// TIA Portal project "Travail_2_station_pince" (V19)

(* hardware
DEVICE "S7-300/ET200M station_1"  S7-300 station
   slot 0: "Rail_0"  Rail  6ES7 390-1***0-0AA0
   slot 2: "PLC_1"  CPU 314C-2 PN/DP  6ES7 314-6EH04-0AB0  V3.3
      slot 2: "PROFINET interface_1"  PN-IO
         slot 1: "Port_1"  Port
         slot 2: "Port_2"  Port
      slot 5: "DI 24/DO 16_1"  DI24/DO16
      slot 6: "AI 5/AO 2_1"  AI5/AO2
      slot 7: "Count_1"  Counter
      slot 8: "Positioning_1"  Positioning
*)

// ===== PLC "PLC_1"  CPU 314C-2 PN/DP =====

VAR_GLOBAL   // PLC tag table "Default tag table"
   "PART_AV" AT %I136.0 : Bool;   // Piece disponible
   "1B1" AT %I136.1 : Bool;   // Préhenseur du magasin gauche (G)
   "1B2" AT %I136.2 : Bool;   // Préhenseur du magasin droit (C)
   "1B3" AT %I136.3 : Bool;   // Préhenseur entrée pieces (D)
   "2B1" AT %I136.4 : Bool;   // Pince sortie (psosition basse)
   "2B2" AT %I136.5 : Bool;   // Pince rentrée (position haute)
   "3B1" AT %I136.6 : Bool;   // Piece dans pince pas noir
   "IP_FI" AT %I136.7 : Bool;   // Station suivante libre
   "Start" AT %I137.0 : Bool;
   "Stop" AT %I137.1 : Bool;
   "Auto/Manu" AT %I137.2 : Bool;
   "Reset" AT %I137.3 : Bool;
   "Emergency Stop" AT %I137.5 : Bool;
   "1M1" AT %Q136.0 : Bool;   // Déplacment préhenseur -> gauche
   "1M2" AT %Q136.1 : Bool;   // Déplacment préhenseur -> droite
   "2M1" AT %Q136.2 : Bool;   // Descente pince
   "3M1" AT %Q136.3 : Bool;   // Ouverture pince
   "IP_N_FO" AT %Q136.7 : Bool;   // Sation occupée
   "Mem_presence_piece_Bus_Asi" AT %M137.0 : Bool;
   "Mem_station_Processing_FREE" AT %M137.1 : Bool;
   "piece_envoyé" AT %M137.2 : Bool;
   "piece_recu" AT %M137.3 : Bool;
END_VAR

DATA_BLOCK "Handling_DB"   // DB1
{ S7_Optimized_Access := 'FALSE' }
VERSION : 0.1
// stored: InstanceOfName Handling
"Handling"
BEGIN
END_DATA_BLOCK

FUNCTION_BLOCK "Handling"   // FB1, GRAPH
{ S7_Optimized_Access := 'FALSE' }
VERSION : 0.1
   VAR_INPUT
      OFF_SQ : Bool := false;   // Turn sequence off
      INIT_SQ : Bool := false;   // Set sequence to initial state
      ACK_EF : Bool := false;   // Acknowledge all errors and faults
      S_PREV : Bool := false;   // Output previous step in parameter S_NO
      S_NEXT : Bool := false;   // Indicate next step in parameter S_NO
      SW_AUTO : Bool := false;   // Automatic mode
      SW_TAP : Bool := false;   // Semiautomatic/switch with transition
      SW_TOP : Bool := false;   // Semiautomatic/ignore transition
      SW_MAN : Bool := false;   // Manual mode
      S_SEL : Int := 0;   // Select step to be output to S_NO
      S_ON : Bool := false;   // Activate step indicated in S_NO
      S_OFF : Bool := false;   // Disable step indicated in S_NO
      T_PUSH : Bool := false;   // Enable transition to switch in semi automatic mode
   END_VAR
   VAR_OUTPUT
      S_NO : Int := 0;   // Step number
      S_MORE : Bool := false;   // More steps are available and can be shown in S_NO
      S_ACTIVE : Bool := false;   // Step indicated in S_NO is active
      ERR_FLT : Bool := false;   // Interlock or supervision group error
      AUTO_ON : Bool := false;   // Automatic mode is active
      TAP_ON : Bool := false;   // Semiautomatic mode/step with transition enabled
      TOP_ON : Bool := false;   // Semiautomatic mode/ignore transition enabled
      MAN_ON : Bool := false;   // Manual mode is active
   END_VAR
   VAR
      SWITCH : Array[0..0] of DWord;
      SW_SQTS : Array[0..19] of Byte;
      SW_ADDR : Word := 16#A;
      G7T_0 : GraphTransition;
      G7S_0 : GraphStep;
      PRE_CRIT : Array[0..0] of DWord;
      POST_CRIT : Array[0..0] of DWord;
      TVX : Array[0..2] of Byte;
      TTX : Array[0..2] of Byte;
      TSX : Array[0..2] of Byte;
      S00X : Array[0..2] of Byte;
      SOFFX : Array[0..2] of Byte;
      SONX : Array[0..2] of Byte;
      SAX : Array[0..2] of Byte;
      SERRX : Array[0..20] of Byte;
      SMX : Array[0..20] of Byte;
      S0X : Array[0..20] of Byte;
      S1X : Array[0..20] of Byte;
      S_DISPLAY : Int;   // Internal display of output parameter S_NO
      S_SEL_OLD : Int;   // Previous value in S_SEL
      S_DISPIDX : Byte;   // Index of the step in S_NO
      T_DISPIDX : Byte;   // Index of the transition displayed in T_NO
      MOPEDGE : Struct
         AUTO : Bool := false;
         MAN : Bool := false;
         TAP : Bool := false;
         TOP : Bool := false;
         ACK_S : Bool := false;
         REG_S : Bool := false;
         T_PREV : Bool := false;
         T_NEXT : Bool := false;
         LOCK : Bool := false;
         SUP : Bool := false;
         ACKREQ : Bool := false;
         SSKIP : Bool := false;
         OFF : Bool := false;
         INIT : Bool := false;
         HALT : Bool := false;
         TMS_HALT : Bool := false;
         OPS_ZERO : Bool := false;
         SACT_DISP : Bool := false;
         SEF_DISP : Bool := false;
         SALL_DISP : Bool := false;
         S_PREV : Bool := false;
         S_NEXT : Bool := false;
         S_SELOK : Bool := false;
         S_ON : Bool := false;
         S_OFF : Bool := false;
         T_PUSH : Bool := false;
         REG : Bool := false;
         ACK : Bool := false;
         IL_PERM : Bool := false;
         T_PERM : Bool := false;
         ILP_MAN : Bool := false;
      END_STRUCT;
      MOP : Struct   // Mode
         AUTO : Bool := true;   // Status: automatic mode
         MAN : Bool := false;   // Status: manual mode
         TAP : Bool := false;   // Status: semi automatic/switch with transition
         TOP : Bool := false;   // Status: semi automatic/ignore transition
         ACK_S : Bool := false;   // Request: acknowledge step at parameter S_NO
         REG_S : Bool := false;   // Request: register step indicated in S_NO
         T_PREV : Bool := false;   // Request: output previous valid transition in T_NO
         T_NEXT : Bool := false;   // Request: output next valid transition in T_NO
         LOCK : Bool := true;   // Status: interlocks enabled
         SUP : Bool := true;   // Status: supervisions enabled
         ACKREQ : Bool := true;   // Status: acknowledgment required
         SSKIP : Bool := false;   // Status: "Skip steps" enabled
         OFF : Bool := false;   // Request: deactivate all steps
         INIT : Bool := true;   // Request: set sequence to initial state
         HALT : Bool := false;   // Status: sequence halted
         TMS_HALT : Bool := false;   // Status: all internal timers held
         OPS_ZERO : Bool := false;   // Status: set all operands processed with N, L, D instructions to 0
         SACT_DISP : Bool := true;   // Status: display active steps only
         SEF_DISP : Bool := false;   // Status: display only steps with errors and disrupted steps
         SALL_DISP : Bool := false;   // Status: display all steps
         S_PREV : Bool := false;   // Request: output previous step to S_NO
         S_NEXT : Bool := false;   // Request: Output next step at S_NO parameter
         S_SELOK : Bool := false;   // Request: output step number from S_SEL to S_NO
         S_ON : Bool := false;   // Request: activate step indicated in S_NO
         S_OFF : Bool := false;   // Request: deactivate step at parameter S_NO
         T_PUSH : Bool := false;   // Request: transition switching enabled
         REG : Bool := false;   // Request: register all interlock and supervision errors
         ACK : Bool := false;   // Request: acknowledge all interlock and supervision errors
         IL_PERM : Bool := false;   // Status: permanent processing of all interlocks
         T_PERM : Bool := false;   // Status: permanent processing of all transitions
         ILP_MAN : Bool := false;   // Status: permanent processing of all interlocks in manual mode
      END_STRUCT;
      TICKS : Struct   // Clock speeds
         DELTA : Time := T#0ms;   // Time difference between two cycles
         OLD : Time := T#0ms;   // 10 ms clock counter value in last cycle
         NEW : Time := T#0ms;   // 10 ms clock counter value in this cycle
      END_STRUCT;
      SQ_FLAGS : Struct   // Sequence bit memory
         ERR_FLT : Bool := false;   // Interlock and supervision group error
         ERROR : Bool := false;   // Interlock group error
         FAULT : Bool := false;   // Supervision group error
         RT_FAIL : Bool := false;   // Runtime error
         NO_SNO : Bool := false;   // Requested step number not found
         NF_OFL : Bool := false;   // Overflow: too many ON or OFF requests
         SA_OFL : Bool := false;   // Overflow: too many steps active
         TV_OFL : Bool := false;   // Overflow: too many valid transitions
         MSG_OFL : Bool := false;   // Overflow: not enough system resources for ALARM_S
         NO_SWI : Bool := false;   // Do not switch in this cycle
         CYC_OP : Bool := false;   // Cyclic execution of the sequence after initialization
         AS_MSG : Bool := true;   // Alarms during runtime enabled or disabled by instruction
         AS_SEND : Bool := false;   // Send alarms from WR_USMSG or only enter in diagnostics buffer
         SQ_BUSY : Bool := false;   // Internal edge bit memory for sequence processing
         SA_BUSY : Bool := false;   // Internal edge bit memory for sequence processing
         AS_SIG : Bool := false;   // Edge bit memory for alarms from Alarm_S and Alarm_SQ
      END_STRUCT;
      S_PTR : DWord := 16#B20;
      S_PTR2 : DWord := 16#0;
      S_PTR3 : DWord := 16#2250;
      S_PTR4 : DWord := 16#21A0;
      T_PTR : DWord := 16#20F0;
      C_AR2 : DWord := 16#0;
      M_FBDB : DWord := 16#10000;
      M_SNO : Word := 16#0;
      M_EVID : Word := 16#0;
      M_EVIL : C_Alarm_s;
      M_EVSV : C_Alarm_s;
      M_EV : DWord := 16#1FE0;
      CRIT : Array[0..31] of Bool;
      S_START : Byte := 16#0;
      S_IDX : Byte := 16#0;
      S_INT : Int := 72;
      S_TMP : Byte := 16#0;
      T_START : Byte := 16#0;
      T_IDX : Byte := 16#0;
      T_TMP : Byte := 16#0;
      T_TMP2 : Byte := 16#00;
      TV_POT : Byte := 16#06;
      RETURN1 : Byte := 16#0;
      RETURN2 : Byte := 16#0;
      SINI : Array[0..2] of Byte;
      LSTT : Array[0..19] of Byte;
      ATAJ : Array[0..19] of Byte;
      ATAB : Array[0..19] of Byte;
      PSTT : Array[0..19] of Byte;
      NSTT : Array[0..19] of Byte;
      ASSJ : Array[0..19] of Byte;
      ASSB : Array[0..19] of Byte;
      PTTS : Array[0..19] of Byte;
      NTTS : Array[0..19] of Byte;
      PRE_CNT : Word := 16#1;
      POST_CNT : Word := 16#1;
      ADR_COND : Word := 16#0;
      MAX_TVAL : Byte := 16#1;
      MAX_SACT : Byte := 16#1;
      MAX_CRIT : Byte := 16#4;
      T_CNT : Byte := 16#13;
      SUP_CNT : Byte := 16#0;
      LOCK_CNT : Byte := 16#0;
      S_CNT : Byte := 16#13;
      SQ_CNT : Byte := 16#1;
      PRS_INPAR : DWord := 16#E000FEC8;
      PRS_OUTPAR : DWord := 16#E000800F;
      GC_FLAGS : Struct
         T_MACH : Byte := 16#EB;
         COND_ED : Byte := 16#E3;
         W_LEVEL : Byte := 16#D5;
         FB_IF : Byte := 16#FA;
         AS_MSG : Word := 16#404;
         SSB : Word := 16#108;
         DILG : Word := 16#598;
         ADDR_T0 : Word := 16#24;
         CRIT_AVAIL : Bool := false;
         SSKIP_AVAIL : Bool := true;
         SSKIP_ON : Bool := false;
         ACK_REQ : Bool := true;
         SYNC_AVAIL : Bool := true;
         ILP_MAN : Bool := false;
         SWM_LOCKED : Bool := false;
         SAVE_SW : Bool := true;
      END_STRUCT;
      G7_FBMARK : Byte := 16#3C;
      G7_RELEASE : Byte := 16#3C;
      G7_ID2 : Byte := 16#37;
      G7_ID1 : Byte := 16#47;
   END_VAR
   // SW_SQTS[0] := 16#1;
   // TVX[0] := 16#1;
   // TTX[0] := 16#1;
   // TSX[0] := 16#1;
   // S00X[0] := 16#1;
   // SOFFX[0] := 16#1;
   // SONX[0] := 16#1;
   // SAX[0] := 16#1;
   // SERRX[0] := 16#1;
   // SMX[0] := 16#1;
   // S0X[0] := 16#1;
   // S1X[0] := 16#1;
   // SINI[0] := 16#2;
   // SINI[1] := 16#1;
   // SINI[2] := 0;
   // LSTT[0] := 0;
   // LSTT[1] := 0;
   // LSTT[2] := 0;
   // LSTT[3] := 0;
   // LSTT[4] := 0;
   // LSTT[5] := 0;
   // LSTT[6] := 0;
   // LSTT[7] := 0;
   // LSTT[8] := 0;
   // LSTT[9] := 0;
   // LSTT[10] := 0;
   // LSTT[11] := 0;
   // LSTT[12] := 0;
   // LSTT[13] := 0;
   // LSTT[14] := 0;
   // LSTT[15] := 0;
   // LSTT[16] := 0;
   // LSTT[17] := 0;
   // LSTT[18] := 0;
   // LSTT[19] := 16#1;
   // ATAJ[0] := 0;
   // ATAJ[1] := 16#1;
   // ATAJ[2] := 16#2;
   // ATAJ[3] := 16#3;
   // ATAJ[4] := 16#4;
   // ATAJ[5] := 16#5;
   // ATAJ[6] := 16#6;
   // ATAJ[7] := 16#7;
   // ATAJ[8] := 16#8;
   // ATAJ[9] := 16#9;
   // ATAJ[10] := 16#A;
   // ATAJ[11] := 16#B;
   // ATAJ[12] := 16#C;
   // ATAJ[13] := 16#D;
   // ATAJ[14] := 16#E;
   // ATAJ[15] := 16#F;
   // ATAJ[16] := 16#10;
   // ATAJ[17] := 16#11;
   // ATAJ[18] := 16#12;
   // ATAJ[19] := 16#13;
   // ATAB[0] := 0;
   // ATAB[1] := 16#1;
   // ATAB[2] := 16#2;
   // ATAB[3] := 16#3;
   // ATAB[4] := 16#4;
   // ATAB[5] := 16#5;
   // ATAB[6] := 16#6;
   // ATAB[7] := 16#7;
   // ATAB[8] := 16#8;
   // ATAB[9] := 16#9;
   // ATAB[10] := 16#A;
   // ATAB[11] := 16#B;
   // ATAB[12] := 16#C;
   // ATAB[13] := 16#D;
   // ATAB[14] := 16#E;
   // ATAB[15] := 16#F;
   // ATAB[16] := 16#10;
   // ATAB[17] := 16#11;
   // ATAB[18] := 16#12;
   // ATAB[19] := 16#13;
   // PSTT[0] := 0;
   // PSTT[1] := 16#1;
   // PSTT[2] := 16#2;
   // PSTT[3] := 16#3;
   // PSTT[4] := 16#4;
   // PSTT[5] := 16#5;
   // PSTT[6] := 16#6;
   // PSTT[7] := 16#7;
   // PSTT[8] := 16#8;
   // PSTT[9] := 16#9;
   // PSTT[10] := 16#A;
   // PSTT[11] := 16#B;
   // PSTT[12] := 16#C;
   // PSTT[13] := 16#D;
   // PSTT[14] := 16#E;
   // PSTT[15] := 16#F;
   // PSTT[16] := 16#10;
   // PSTT[17] := 16#11;
   // PSTT[18] := 16#12;
   // PSTT[19] := 16#13;
   // NSTT[0] := 16#1;
   // NSTT[1] := 16#2;
   // NSTT[2] := 16#3;
   // NSTT[3] := 16#4;
   // NSTT[4] := 16#5;
   // NSTT[5] := 16#6;
   // NSTT[6] := 16#7;
   // NSTT[7] := 16#8;
   // NSTT[8] := 16#9;
   // NSTT[9] := 16#A;
   // NSTT[10] := 16#B;
   // NSTT[11] := 16#C;
   // NSTT[12] := 16#D;
   // NSTT[13] := 16#E;
   // NSTT[14] := 16#F;
   // NSTT[15] := 16#10;
   // NSTT[16] := 16#11;
   // NSTT[17] := 16#12;
   // NSTT[18] := 16#13;
   // NSTT[19] := 16#1;
   // ASSJ[0] := 0;
   // ASSJ[1] := 16#1;
   // ASSJ[2] := 16#2;
   // ASSJ[3] := 16#3;
   // ASSJ[4] := 16#4;
   // ASSJ[5] := 16#5;
   // ASSJ[6] := 16#6;
   // ASSJ[7] := 16#7;
   // ASSJ[8] := 16#8;
   // ASSJ[9] := 16#9;
   // ASSJ[10] := 16#A;
   // ASSJ[11] := 16#B;
   // ASSJ[12] := 16#C;
   // ASSJ[13] := 16#D;
   // ASSJ[14] := 16#E;
   // ASSJ[15] := 16#F;
   // ASSJ[16] := 16#10;
   // ASSJ[17] := 16#11;
   // ASSJ[18] := 16#12;
   // ASSJ[19] := 16#13;
   // ASSB[0] := 0;
   // ASSB[1] := 16#1;
   // ASSB[2] := 16#2;
   // ASSB[3] := 16#3;
   // ASSB[4] := 16#4;
   // ASSB[5] := 16#5;
   // ASSB[6] := 16#6;
   // ASSB[7] := 16#7;
   // ASSB[8] := 16#8;
   // ASSB[9] := 16#9;
   // ASSB[10] := 16#A;
   // ASSB[11] := 16#B;
   // ASSB[12] := 16#C;
   // ASSB[13] := 16#D;
   // ASSB[14] := 16#E;
   // ASSB[15] := 16#F;
   // ASSB[16] := 16#10;
   // ASSB[17] := 16#11;
   // ASSB[18] := 16#12;
   // ASSB[19] := 16#13;
   // PTTS[0] := 0;
   // PTTS[2] := 16#1;
   // PTTS[3] := 16#2;
   // PTTS[4] := 16#3;
   // PTTS[5] := 16#4;
   // PTTS[6] := 16#5;
   // PTTS[7] := 16#6;
   // PTTS[8] := 16#7;
   // PTTS[9] := 16#8;
   // PTTS[10] := 16#9;
   // PTTS[11] := 16#A;
   // PTTS[12] := 16#B;
   // PTTS[13] := 16#C;
   // PTTS[14] := 16#D;
   // PTTS[15] := 16#E;
   // PTTS[16] := 16#F;
   // PTTS[17] := 16#10;
   // PTTS[18] := 16#11;
   // PTTS[19] := 16#12;
   // NTTS[0] := 0;
   // NTTS[1] := 16#1;
   // NTTS[2] := 16#2;
   // NTTS[3] := 16#3;
   // NTTS[4] := 16#4;
   // NTTS[5] := 16#5;
   // NTTS[6] := 16#6;
   // NTTS[7] := 16#7;
   // NTTS[8] := 16#8;
   // NTTS[9] := 16#9;
   // NTTS[10] := 16#A;
   // NTTS[11] := 16#B;
   // NTTS[12] := 16#C;
   // NTTS[13] := 16#D;
   // NTTS[14] := 16#E;
   // NTTS[15] := 16#F;
   // NTTS[16] := 16#10;
   // NTTS[17] := 16#11;
   // NTTS[18] := 16#12;
   // NTTS[19] := 16#13;
BEGIN
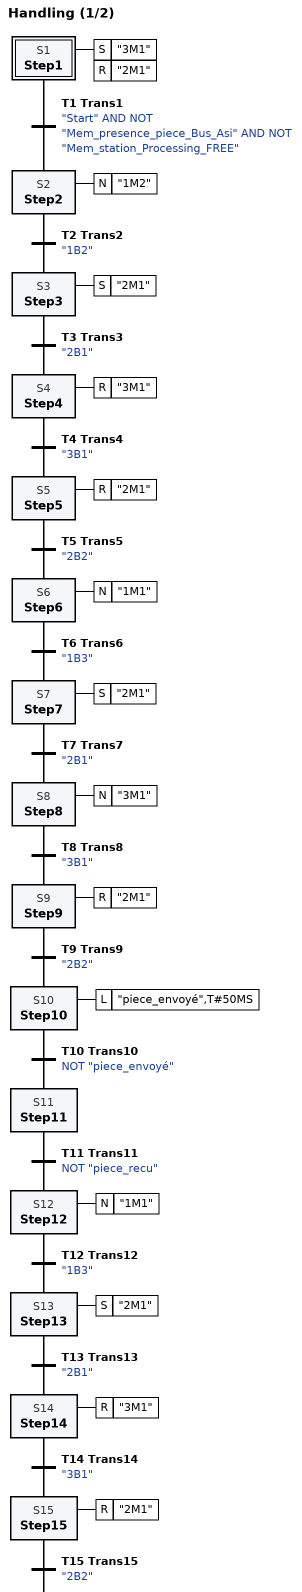
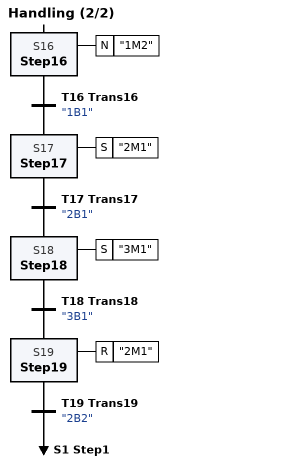
   // sequencer 1
   INITIAL_STEP Step1:   // S1
              S    "3M1"
              R    "2M1"
   END_STEP
   TRANSITION Trans1 FROM Step1 TO Step2   // T1
      := "Start" AND NOT "Mem_presence_piece_Bus_Asi" AND NOT "Mem_station_Processing_FREE";
   END_TRANSITION
   STEP Step2:   // S2
              N    "1M2"
   END_STEP
   TRANSITION Trans2 FROM Step2 TO Step3   // T2
      := "1B2";
   END_TRANSITION
   STEP Step3:   // S3
              S    "2M1"
   END_STEP
   TRANSITION Trans3 FROM Step3 TO Step4   // T3
      := "2B1";
   END_TRANSITION
   STEP Step4:   // S4
              R    "3M1"
   END_STEP
   TRANSITION Trans4 FROM Step4 TO Step5   // T4
      := "3B1";
   END_TRANSITION
   STEP Step5:   // S5
              R    "2M1"
   END_STEP
   TRANSITION Trans5 FROM Step5 TO Step6   // T5
      := "2B2";
   END_TRANSITION
   STEP Step6:   // S6
              N    "1M1"
   END_STEP
   TRANSITION Trans6 FROM Step6 TO Step7   // T6
      := "1B3";
   END_TRANSITION
   STEP Step7:   // S7
              S    "2M1"
   END_STEP
   TRANSITION Trans7 FROM Step7 TO Step8   // T7
      := "2B1";
   END_TRANSITION
   STEP Step8:   // S8
              N    "3M1"
   END_STEP
   TRANSITION Trans8 FROM Step8 TO Step9   // T8
      := "3B1";
   END_TRANSITION
   STEP Step9:   // S9
              R    "2M1"
   END_STEP
   TRANSITION Trans9 FROM Step9 TO Step10   // T9
      := "2B2";
   END_TRANSITION
   STEP Step10:   // S10
              L    "piece_envoyé",T#50MS
   END_STEP
   TRANSITION Trans10 FROM Step10 TO Step11   // T10
      := NOT "piece_envoyé";
   END_TRANSITION
   STEP Step11:   // S11
   END_STEP
   TRANSITION Trans11 FROM Step11 TO Step12   // T11
      := NOT "piece_recu";
   END_TRANSITION
   STEP Step12:   // S12
              N    "1M1"
   END_STEP
   TRANSITION Trans12 FROM Step12 TO Step13   // T12
      := "1B3";
   END_TRANSITION
   STEP Step13:   // S13
              S    "2M1"
   END_STEP
   TRANSITION Trans13 FROM Step13 TO Step14   // T13
      := "2B1";
   END_TRANSITION
   STEP Step14:   // S14
              R    "3M1"
   END_STEP
   TRANSITION Trans14 FROM Step14 TO Step15   // T14
      := "3B1";
   END_TRANSITION
   STEP Step15:   // S15
              R    "2M1"
   END_STEP
   TRANSITION Trans15 FROM Step15 TO Step16   // T15
      := "2B2";
   END_TRANSITION
   STEP Step16:   // S16
              N    "1M2"
   END_STEP
   TRANSITION Trans16 FROM Step16 TO Step17   // T16
      := "1B1";
   END_TRANSITION
   STEP Step17:   // S17
              S    "2M1"
   END_STEP
   TRANSITION Trans17 FROM Step17 TO Step18   // T17
      := "2B1";
   END_TRANSITION
   STEP Step18:   // S18
              S    "3M1"
   END_STEP
   TRANSITION Trans18 FROM Step18 TO Step19   // T18
      := "3B1";
   END_TRANSITION
   STEP Step19:   // S19
              R    "2M1"
   END_STEP
   TRANSITION Trans19 FROM Step19 TO Step1   // T19, jump
      := "2B2";
   END_TRANSITION
END_FUNCTION_BLOCK

ORGANIZATION_BLOCK "Main"   // OB1, LAD
TITLE = "Main Program Sweep (Cycle)"
{ S7_Optimized_Access := 'FALSE' }
VERSION : 0.1
   VAR_TEMP
      OB1_EV_CLASS : Byte;   // Bits 0-3 = 1 (Coming event), Bits 4-7 = 1 (Event class 1)
      OB1_SCAN_1 : Byte;   // 1 (Cold restart scan 1 of OB 1), 3 (Scan 2-n of OB 1)
      OB1_PRIORITY : Byte;   // Priority of OB Execution
      OB1_OB_NUMBR : Byte;   // 1 (Organization block 1, OB1)
      OB1_RESERVED_1 : Byte;   // Reserved for system
      OB1_RESERVED_2 : Byte;   // Reserved for system
      OB1_PREV_CYCLE : Int;   // Cycle time of previous OB1 scan (milliseconds)
      OB1_MIN_CYCLE : Int;   // Minimum cycle time of OB1 (milliseconds)
      OB1_MAX_CYCLE : Int;   // Maximum cycle time of OB1 (milliseconds)
      OB1_DATE_TIME : Date_And_Time;   // Date and time OB1 started
   END_VAR
BEGIN

REGION Network 1
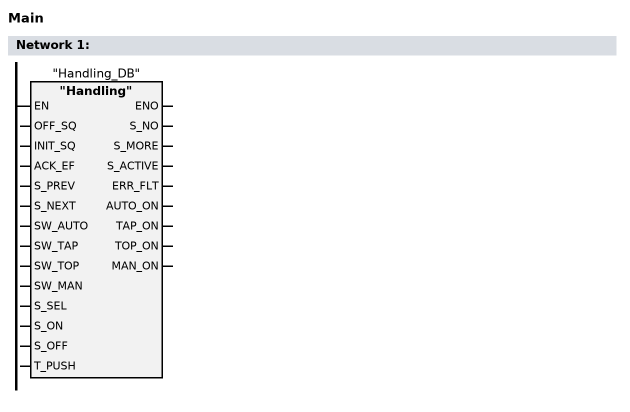
   RUNG wire#powerrail
      "Handling_DB"(OFF_SQ :=, INIT_SQ :=, ACK_EF :=, S_PREV :=, S_NEXT :=, SW_AUTO :=, SW_TAP :=, SW_TOP :=, SW_MAN :=, S_SEL :=, S_ON :=, S_OFF :=, T_PUSH :=, S_NO =>, S_MORE =>, S_ACTIVE =>, ERR_FLT =>, AUTO_ON =>, TAP_ON =>, TOP_ON =>, MAN_ON =>)
   END_RUNG
   // the same network as SCL:
   "Handling_DB"();   // "Handling"
END_REGION
END_ORGANIZATION_BLOCK